{attribute 'qualified_only'}
VAR_GLOBAL
	TuerAuf : BOOL;
	TuerZu : BOOL;
	AktuellerStock : INT;
	
END_VAR

(* stored: Version 1.1.0.1
   GVL Visu_Liftkabine: Id {bcd6e263-cee3-49d0-a165-a4d6b1cba7ae} *)
